FUNCTION_BLOCK FB_HybridDispenser EXTENDS FB_GCodeTool IMPLEMENTS I_Dispenser
VAR_INPUT
END_VAR
VAR_OUTPUT
END_VAR
VAR
	//Specproperties
	aiDispenser		: ARRAY[1..3] OF I_Dispenser;
	nMasterSlotNr	: USINT;

	//****************************************Aktionsvariablen****************************************************
	bBasicDispense			: BOOL;
	nStateA_BasicDispense 	: USINT;
	
	n : INT; //Zählvariablen
	m : INT; //Zählvariablen

END_VAR

IF eCurrentState = E_MachineState.MACHINESTATE_Active THEN
	IF bBasicDispense THEN
		A_HybridDispense();
		IF nStateA_BasicDispense >= 80 THEN
			IF nStateA_BasicDispense >= 99 THEN
				bError := TRUE;
			END_IF
			bBasicDispense := FALSE;
			nStateA_BasicDispense := 0;
			M_RemoveListEntry(nSearchValue:= E_Action.ACTION_BasicDispense);
		END_IF
	END_IF
END_IF

SUPER^();	//FB_MzTool aufrufen

//Prozessdaten aktualisieren
stProcessData.n32Data[7] := BOOL_TO_DINT(bBasicDispense);
aObjProcData[nNotifyId] := stProcessData;

ACTION A_HybridDispense:
IF nStateA_BasicDispense = 0 THEN	//alle Dispenser starten
	FOR n := 1 TO 3 BY 1 DO
		IF aiDispenser[n] <> 0 THEN
			stError.ErrorId := aiDispenser[n].M_DispenserStart();
			stError.ObjectId := aiDispenser[n].P_pObject^.P_nObjectID;
			IF stError.ErrorId > 0 THEN
				//Bereits gestartete Tools wieder stoppen
				FOR m := 1 TO n - 1 BY 1 DO
					aiDispenser[m].M_DispenserStop();
				END_FOR
				nStateA_BasicDispense := 99;
				EXIT;
			END_IF
		END_IF
	END_FOR
	IF nStateA_BasicDispense = 0 THEN
		nStateA_BasicDispense := 1;	
	END_IF
END_IF

IF nStateA_BasicDispense = 1 THEN	//alle Dispenser laufen -> permanent auf Fehler überwachen
	//Das Verlassen dieses States erfolgt durch die Action "HybridDispense" mit Parameter "off" oder durch Stop bzw. Cancel
	FOR n := 1 TO 3 BY 1 DO
		IF aiDispenser[n] <> 0 THEN
			IF aiDispenser[n].P_bError THEN
				stError.ErrorId := aiDispenser[n].P_nErrorId;
				stError.ObjectId := aiDispenser[n].P_pObject^.P_nObjectID;
				nStateA_BasicDispense := 2; //weiter zu stoppen
				EXIT;
			END_IF
		END_IF
	END_FOR	
END_IF

IF nStateA_BasicDispense = 2 THEN //übrige Dispenser nach Fehler stoppen
	nStateA_BasicDispense := 99;
	FOR n := 1 TO 3 BY 1 DO
		IF aiDispenser[n] <> 0 THEN
			IF NOT aiDispenser[n].P_bError THEN
				aiDispenser[n].M_DispenserStop();
			END_IF
		END_IF
	END_FOR	
END_IF

IF nStateA_BasicDispense = 70 THEN //Dispenser stoppen
	nStateA_BasicDispense := 71;
	FOR n := 1 TO 3 BY 1 DO
		IF aiDispenser[n] <> 0 THEN
			aiDispenser[n].M_DispenserStop();
		END_IF
	END_FOR	
ELSIF nStateA_BasicDispense = 71 THEN //warten bis alle Dispenser gestoppt
	nStateA_BasicDispense := 80;
	FOR n := 1 TO 3 BY 1 DO
		IF aiDispenser[n] <> 0 THEN
			IF NOT aiDispenser[n].P_eDispenserState = E_DispenserState.Idle THEN 
				nStateA_BasicDispense := 71;
			END_IF
		END_IF
	END_FOR	
END_IF

//Errorhandling
IF nStateA_BasicDispense = 99 THEN
	stError.Cmd := E_Action.ACTION_BasicDispense;
	stError.POU := E_POU.POU_FB_HybridDispenser;
	stError.POUAction := E_POUACT.POUACT_A_BasicDispense;
	fbErrorList.M_Add(stError);
END_IF
END_ACTION

ACTION A_Reset:
//Ist noch eine Aktion aktiv?
IF nStateA_ResetSpec = 0 THEN 
	(*IF bHeating THEN
		bHeating := FALSE;
		nStateA_Heating := 0;
	END_IF*)
	nStateA_ResetSpec := 80;
END_IF

SUPER^.A_Reset();
END_ACTION

ACTION A_Stop:
IF nStateA_Stop = 0 THEN
	IF bBasicDispense AND nStateA_BasicDispense = 1 THEN
		nStateA_BasicDispense := 70;
	END_IF
	nStateA_Stop := 1;	
END_IF

SUPER^.A_Stop();
END_ACTION

METHOD FB_init : BOOL
VAR_INPUT
	bInitRetains : BOOL; // if TRUE, the retain variables are initialized (warm start / cold start)
	bInCopyCode : BOOL;  // if TRUE, the instance afterwards gets moved into the copy code (online change)
END_VAR
eObjectType := E_ObjectType.OBJECTTYPE_HybridDispenser;
eObjectGroup := E_ObjectGroup.OBJECTGROUP_MzTool OR E_ObjectGroup.OBJECTGROUP_Device;
END_METHOD

METHOD M_AddChild : ERRORID
VAR_INPUT
	pObject : POINTER TO FB_Object;
	nSlotNr	: UINT;
	nIndex : INT;
END_VAR
//Der HybridDispenser kann folgende Objekttypen aufnehmen
//Extruder, PassivePip, CartDispenser
IF pObject > 0 THEN
	IF pObject^.P_eObjectType = E_ObjectType.OBJECTTYPE_Extruder OR
		pObject^.P_eObjectType = E_ObjectType.OBJECTTYPE_CartDispenser OR
		pObject^.P_eObjectType = E_ObjectType.OBJECTTYPE_CartDispStirrer OR
		pObject^.P_eObjectType = E_ObjectType.OBJECTTYPE_PassivPip THEN
		M_AddChild := SUPER^.M_AddChild(pObject,nSlotNr,nIndex);
	ELSE
		M_AddChild := E_ErrorIdObjMgmt.ERRORID_InvalidParentObject;
	END_IF
ELSE
	M_AddChild := E_ErrorIdObjMgmt.ERRORID_InvalidParentObject;
END_IF
END_METHOD

METHOD M_CancelAction
VAR_INPUT
	eAction : E_Action;
END_VAR
CASE eAction OF
	E_Action.ACTION_BasicDispense:
		IF bBasicDispense AND nStateA_BasicDispense = 1 THEN
			nStateA_BasicDispense := 70;
		END_IF
ELSE
	SUPER^.M_CancelAction(eAction);
END_CASE
END_METHOD

METHOD M_CheckAction : ERRORID
VAR_INPUT
	refActionData 	: REFERENCE TO ST_ActionData;
	pCorrelObject	: POINTER TO FB_Object;
END_VAR
CASE refActionData.eAction OF
	E_Action.ACTION_Dispense,
	E_Action.ACTION_CleanTip,
	E_Action.ACTION_MeasureTool,
	E_Action.ACTION_TeachTarget:
		RETURN;
ELSE
	M_CheckAction := SUPER^.M_CheckAction(refActionData, pCorrelObject);
END_CASE
END_METHOD

METHOD M_CheckGCodeStart : ERRORID
VAR_INPUT
END_VAR

VAR
	i : USINT;
	pGCodeTool : POINTER TO FB_GCodeTool;
END_VAR
FOR i := 1 TO 3 BY 1 DO
	IF aiDispenser[i] <> 0 AND_THEN aiDispenser[i].P_pObject^.P_eObjectType = E_ObjectType.OBJECTTYPE_Extruder THEN
		pGCodeTool := aiDispenser[i].P_pObject;
		M_CheckGCodeStart := pGCodeTool^.M_CheckGCodeStart();
		IF M_CheckGCodeStart > 0 THEN
			RETURN;
		END_IF
	END_IF
END_FOR
END_METHOD

METHOD M_CheckProcDataType : BOOL
VAR_INPUT
	eProcDataType : E_ProcDataType;
END_VAR
END_METHOD

METHOD M_CheckProps : ERRORID
VAR_INPUT
END_VAR

VAR
	i 				: UINT;
	pSlot 			: POINTER TO FB_Slot;
	pExtruder 		: POINTER TO FB_Extruder;
	pCartDispenser 	: POINTER TO FB_CartDispenser;
	pPassivePip 	: POINTER TO FB_PassivPip;
END_VAR
M_CheckProps := SUPER^.M_CheckProps();
//Kann bis zu 3 CartDispenser enthalten
aiDispenser[1] := 0;
aiDispenser[2] := 0;
aiDispenser[3] := 0;
FOR i:= 1 TO nNumberOfSlots BY 1 DO
	pSlot := fbSlotList.M_GetAtNr(i);
	IF pSlot > 0 AND_THEN pSlot^.P_pChild > 0  THEN
		//Achtung, nur Tools die das Interface "I_HybridDispenser" implementieren sind erlaubt!
		IF pSlot^.P_pChild^.P_eObjectType = E_ObjectType.OBJECTTYPE_Extruder THEN
			pExtruder := pSlot^.P_pChild;
			aiDispenser[pSlot^.P_nNr] := pExtruder^;
		ELSIF pSlot^.P_pChild^.P_eObjectType = E_ObjectType.OBJECTTYPE_CartDispenser OR 
				pSlot^.P_pChild^.P_eObjectType = E_ObjectType.OBJECTTYPE_CartDispStirrer THEN
			pCartDispenser := pSlot^.P_pChild;
			aiDispenser[pSlot^.P_nNr] := pCartDispenser^;
		ELSIF pSlot^.P_pChild^.P_eObjectType = E_ObjectType.OBJECTTYPE_PassivPip THEN
			pPassivePip := pSlot^.P_pChild;
			aiDispenser[pSlot^.P_nNr] := pPassivePip^;
		END_IF
	END_IF
END_FOR
//MasterSlotNr auswerten
//1. kann nur 1,2 oder 3 sein
//2. entsprechender Slot muss belegt sein
IF nMasterSlotNr >= 1 AND nMasterSlotNr <= 3 THEN
	IF aiDispenser[nMasterSlotNr] = 0 THEN
		M_CheckProps := E_ErrorIdObjMgmt.ERRORID_NoToolOnMasterSlot;	
	END_IF
ELSE
	M_CheckProps := E_ErrorIdObjMgmt.ERRORID_InvalidSlotNumber;
END_IF
END_METHOD

METHOD M_ClearAllProps
VAR_INPUT
	bIgnoreParent : BOOL; //Es wird das gesamte OD gelöscht. -> Zeiger auf Parent nicht mehr gültig!
END_VAR
aiDispenser[1] := 0;
aiDispenser[2] := 0;
aiDispenser[3] := 0;
SUPER^.M_ClearAllProps(bIgnoreParent);
END_METHOD

METHOD M_DispenserPrepare : ERRORID
VAR_INPUT
END_VAR
//do nothing
END_METHOD

METHOD M_DispenserStart : ERRORID
VAR_INPUT
END_VAR
IF NOT (eCurrentState = E_MachineState.MACHINESTATE_Idle OR
	eCurrentState = E_MachineState.MACHINESTATE_Active OR
	eCurrentState = E_MachineState.MACHINESTATE_Ready) THEN
	M_DispenserStart := E_ErrorIdCmd.ERRORID_InvalidState;
	RETURN;
END_IF
			
IF NOT bBasicDispense THEN
	bBasicDispense := TRUE;
	fbList.A_AddHeadValue(hList := hList, putValue := E_Action.ACTION_BasicDispense);
ELSE //Bereits Ein -> Error werfen
	M_DispenserStart := E_ErrorIdCmd.ERRORID_BasicActionActive;
	RETURN;
END_IF

bBusy := TRUE;
eCurrentState := E_MachineState.MACHINESTATE_Active;
END_METHOD

METHOD M_DispenserStop : ERRORID
VAR_INPUT
END_VAR
IF bBasicDispense AND nStateA_BasicDispense = 1 THEN
	nStateA_BasicDispense := 70;
END_IF
END_METHOD

METHOD M_ExeAction : ERRORID
VAR_INPUT
	refActionData : REFERENCE TO ST_ActionData;	
END_VAR
IF NOT (eCurrentState = E_MachineState.MACHINESTATE_Idle OR
	eCurrentState = E_MachineState.MACHINESTATE_Active OR
	eCurrentState = E_MachineState.MACHINESTATE_Ready) THEN
	M_ExeAction := E_ErrorIdCmd.ERRORID_InvalidState;
	RETURN;
END_IF

CASE refActionData.eAction OF
	E_Action.ACTION_BasicDispense:
		IF refActionData.aParams[1] = 0 THEN //Aus
			M_ExeAction := M_DispenserStop();
		ELSE //Ein
			M_ExeAction := M_DispenserStart();
		END_IF
	ELSE
		M_ExeAction := SUPER^.M_ExeAction(refActionData);
		RETURN;
END_CASE
END_METHOD

METHOD M_GetAllProps : ERRORID
VAR_INPUT
	refCmdData : REFERENCE TO  ST_CmdData;
END_VAR
SUPER^.M_GetAllProps(refCmdData);
nCurrentPropIndex := nCurrentPropIndex + 1;
refCmdData.n32Data[nCurrentPropIndex] := nMasterSlotNr;
END_METHOD

METHOD M_GetNozzle : POINTER TO FB_Nozzle
VAR_INPUT
END_VAR
IF P_pMasterTool > 0 THEN
	M_GetNozzle := P_pMasterTool^.M_GetNozzle();
END_IF
END_METHOD

METHOD M_GetProcData : DINT
VAR_INPUT
	eProcDataType : E_ProcDataType;
END_VAR
END_METHOD

METHOD M_GetZAxisRef : POINTER TO FB_ZAxisRef
VAR_INPUT
	pTool : POINTER TO FB_MzTool;
	pToolSlot : POINTER TO FB_Slot;
END_VAR

VAR
	nSlotDiff : INT;
	nAxisNr : INT;
END_VAR
//Diese Methode überschreibt sie Methode von FB_MzTool und wird derzeit nur vom SyringeExtruder (Child) aufgerufen
IF pTool^.P_eObjectType = E_ObjectType.OBJECTTYPE_Extruder THEN
	nSlotDiff :=  UINT_TO_INT(pToolSlot^.P_nNr) - UINT_TO_INT(nMasterSlotNr);
	nAxisNr := pZAxisRef^.nChannel + nSlotDiff * 2; //Es muss immer eine freie Achse dazwischen sein.
	M_GetZAxisRef := ADR(pFbMultiZ^.aFbZAxisRef[nAxisNr]);
	IF M_GetZAxisRef^.eDetectedToolType <> E_MzToolType.TOOL_TYPE_SyringeExtruder THEN
		M_GetZAxisRef := 0;
	END_IF
ELSE
	M_GetZAxisRef := SUPER^.M_GetZAxisRef(pTool, pParentSlot);
END_IF
END_METHOD

METHOD M_Prepare : ST_MethResult
VAR_INPUT
	bExecute : BOOL;
END_VAR

VAR
 	i : USINT;	
END_VAR

VAR_INST
	nState : USINT;	
END_VAR
IF bExecute THEN
	IF nState = 0 THEN
		nState := 80;
		FOR i := 1 TO 3 BY 1 DO
			IF aiDispenser[i] <> 0 THEN
				M_Prepare.nErrorId := aiDispenser[i].M_DispenserPrepare();
				IF M_Prepare.nErrorId > 0 THEN
					M_Prepare.bError := TRUE;
					M_Prepare.bBusy := FALSE;
					RETURN;
				END_IF
				IF aiDispenser[i].P_eDispenserState = E_DispenserState.Preparing THEN
					nState := 1;
					M_Prepare.bBusy := TRUE;				
					RETURN;
				END_IF
			END_IF
		END_FOR
	ELSIF nState = 1 THEN
		FOR i := 1 TO 3 BY 1 DO
			IF aiDispenser[i] <> 0 THEN
				IF aiDispenser[i].P_bError THEN
					M_Prepare.bError := TRUE;
					M_Prepare.bBusy := FALSE;
					RETURN;
				END_IF
				IF aiDispenser[i].P_eDispenserState = E_DispenserState.Preparing THEN
					nState := 1;
					M_Prepare.bBusy := TRUE;
					RETURN;
				END_IF				
			END_IF
		END_FOR
	END_IF
ELSE
	nState := 0;	
END_IF
END_METHOD

METHOD M_SetAllProps : ERRORID
VAR_INPUT
	refCmdData : REFERENCE TO  ST_CmdData;
END_VAR
M_SetAllProps := SUPER^.M_SetAllProps(refCmdData);

IF M_SetAllProps > 0 THEN
	RETURN;
END_IF

nCurrentPropIndex := nCurrentPropIndex + 1;
nSpecPropIndex := nCurrentPropIndex;
nMasterSlotNr := DINT_TO_USINT(refCmdData.n32Data[nCurrentPropIndex]);
nNoOfProps := nCurrentPropIndex + 1;
END_METHOD

METHOD M_SetPrintParams : ST_MethResult
VAR_INPUT
	eType 		: E_PrintParamType;
	nNumerator	: USINT;
	nValue		: DINT;
END_VAR

VAR
	pGCodeTool		: POINTER TO FB_GCodeTool;
END_VAR
CASE eType OF
	E_PrintParamType.Pressure:
		CASE nNumerator OF
			1:	IF aiDispenser[1] <> 0 AND_THEN 
					(aiDispenser[1].P_pObject^.P_eObjectType = E_ObjectType.OBJECTTYPE_CartDispenser OR	aiDispenser[1].P_pObject^.P_eObjectType = E_ObjectType.OBJECTTYPE_CartDispStirrer) THEN
					pGCodeTool := aiDispenser[1].P_pObject;
					M_SetPrintParams := pGCodeTool^.M_SetPrintParams(E_PrintParamType.Pressure, 1, nValue);
				ELSE
					M_SetPrintParams.bError := TRUE;
					M_SetPrintParams.nErrorId := E_ErrorIdCmd.ERRORID_InvalidPrintParamType;
				END_IF
				
			2:	IF aiDispenser[2] <> 0 AND_THEN
					(aiDispenser[2].P_pObject^.P_eObjectType = E_ObjectType.OBJECTTYPE_CartDispenser OR aiDispenser[2].P_pObject^.P_eObjectType = E_ObjectType.OBJECTTYPE_CartDispStirrer) THEN
					pGCodeTool := aiDispenser[2].P_pObject;
					M_SetPrintParams := pGCodeTool^.M_SetPrintParams(E_PrintParamType.Pressure, 1, nValue);
				ELSE
					M_SetPrintParams.bError := TRUE;
					M_SetPrintParams.nErrorId := E_ErrorIdCmd.ERRORID_InvalidPrintParamType;
				END_IF
			
			3: IF aiDispenser[3] <> 0 AND_THEN
					(aiDispenser[3].P_pObject^.P_eObjectType = E_ObjectType.OBJECTTYPE_CartDispenser OR aiDispenser[3].P_pObject^.P_eObjectType = E_ObjectType.OBJECTTYPE_CartDispStirrer) THEN
					pGCodeTool := aiDispenser[3].P_pObject;
					M_SetPrintParams := pGCodeTool^.M_SetPrintParams(E_PrintParamType.Pressure, 1, nValue);
				ELSE
					M_SetPrintParams.bError := TRUE;
					M_SetPrintParams.nErrorId := E_ErrorIdCmd.ERRORID_InvalidPrintParamType;
				END_IF
		ELSE
			M_SetPrintParams.bError := TRUE;
			M_SetPrintParams.nErrorId := E_ErrorIdCmd.ERRORID_InvalidPrintParamNumerator;
		END_CASE
		
	E_PrintParamType.Feed:
		CASE nNumerator OF
			1:	IF aiDispenser[1] <> 0 AND_THEN aiDispenser[1].P_pObject^.P_eObjectType = E_ObjectType.OBJECTTYPE_Extruder THEN
					pGCodeTool := aiDispenser[1].P_pObject;
					M_SetPrintParams := pGCodeTool^.M_SetPrintParams(E_PrintParamType.Feed, 1, nValue);
				ELSE
					M_SetPrintParams.bError := TRUE;
					M_SetPrintParams.nErrorId := E_ErrorIdCmd.ERRORID_InvalidPrintParamType;
				END_IF
			
			2:	IF aiDispenser[2] <> 0 AND_THEN aiDispenser[2].P_pObject^.P_eObjectType = E_ObjectType.OBJECTTYPE_Extruder THEN
					pGCodeTool := aiDispenser[2].P_pObject;
					M_SetPrintParams := pGCodeTool^.M_SetPrintParams(E_PrintParamType.Feed, 1, nValue);
				ELSE
					M_SetPrintParams.bError := TRUE;
					M_SetPrintParams.nErrorId := E_ErrorIdCmd.ERRORID_InvalidPrintParamType;
				END_IF
			
			3:	IF aiDispenser[3] <> 0 AND_THEN aiDispenser[3].P_pObject^.P_eObjectType = E_ObjectType.OBJECTTYPE_Extruder THEN
					pGCodeTool := aiDispenser[3].P_pObject;
					M_SetPrintParams := pGCodeTool^.M_SetPrintParams(E_PrintParamType.Feed, 1, nValue);			
				ELSE
					M_SetPrintParams.bError := TRUE;
					M_SetPrintParams.nErrorId := E_ErrorIdCmd.ERRORID_InvalidPrintParamType;
				END_IF
			
		ELSE
			M_SetPrintParams.bError := TRUE;
			M_SetPrintParams.nErrorId := E_ErrorIdCmd.ERRORID_InvalidPrintParamNumerator;
		END_CASE
		
	E_PrintParamType.Flow:
		CASE nNumerator OF
			1:	IF aiDispenser[1] <> 0 AND_THEN aiDispenser[1].P_pObject^.P_eObjectType = E_ObjectType.OBJECTTYPE_PassivPip THEN
					pGCodeTool := aiDispenser[1].P_pObject;
					M_SetPrintParams := pGCodeTool^.M_SetPrintParams(E_PrintParamType.Flow, 1, nValue);			
				ELSE
					M_SetPrintParams.bError := TRUE;
					M_SetPrintParams.nErrorId := E_ErrorIdCmd.ERRORID_InvalidPrintParamType;
				END_IF
			
			2:	IF aiDispenser[2] <> 0 AND_THEN aiDispenser[2].P_pObject^.P_eObjectType = E_ObjectType.OBJECTTYPE_PassivPip THEN
					pGCodeTool := aiDispenser[2].P_pObject;
					M_SetPrintParams := pGCodeTool^.M_SetPrintParams(E_PrintParamType.Flow, 1, nValue);			
				ELSE
					M_SetPrintParams.bError := TRUE;
					M_SetPrintParams.nErrorId := E_ErrorIdCmd.ERRORID_InvalidPrintParamType;
				END_IF
			
			3:	IF aiDispenser[3] <> 0 AND_THEN aiDispenser[3].P_pObject^.P_eObjectType = E_ObjectType.OBJECTTYPE_PassivPip THEN
					pGCodeTool := aiDispenser[3].P_pObject;
					M_SetPrintParams := pGCodeTool^.M_SetPrintParams(E_PrintParamType.Flow, 1, nValue);
				ELSE
					M_SetPrintParams.bError := TRUE;
					M_SetPrintParams.nErrorId := E_ErrorIdCmd.ERRORID_InvalidPrintParamType;
				END_IF
		ELSE
			M_SetPrintParams.bError := TRUE;
			M_SetPrintParams.nErrorId := E_ErrorIdCmd.ERRORID_InvalidPrintParamNumerator;
		END_CASE
	
ELSE
	M_SetPrintParams.bError := TRUE;
	M_SetPrintParams.nErrorId := E_ErrorIdCmd.ERRORID_InvalidPrintParamType;	
END_CASE
END_METHOD

METHOD M_ToolIsOnMasterSlot : BOOL
VAR_INPUT
	pTool : POINTER TO FB_MzTool;
END_VAR
IF aiDispenser[nMasterSlotNr] <> 0 THEN
	M_ToolIsOnMasterSlot := aiDispenser[nMasterSlotNr].P_pObject = pTool;
END_IF
END_METHOD

PROPERTY P_bSensorMounted : BOOL
GET
VAR
	i : USINT;
	pTool : POINTER TO FB_MzTool;
END_VAR
FOR i := 1 TO 3 BY 1 DO
	IF aiDispenser[i] <> 0 THEN
		pTool := aiDispenser[i].P_pObject;
		IF pTool^.P_bSensorMounted THEN
			P_bSensorMounted := TRUE;
			RETURN;
		END_IF
	END_IF
END_FOR
END_GET
END_PROPERTY

PROPERTY P_eDispenserState : E_DispenserState
GET
IF bBasicDispense THEN
	//falls ein Dispenser in Preparing ist, dann bleibt es auch so
	P_eDispenserState := E_DispenserState.Dispensing;
END_IF
END_GET
END_PROPERTY

PROPERTY P_pMasterTool : POINTER TO FB_MzTool
GET
P_pMasterTool := aiDispenser[nMasterSlotNr].P_pObject;
END_GET
END_PROPERTY

PROPERTY P_stAbsPosPhys : ST_3DPoint
GET
VAR
	pMzTool : POINTER TO FB_MzTool;
END_VAR
IF aiDispenser[nMasterSlotNr] <> 0 THEN
	pMzTool := aiDispenser[nMasterSlotNr].P_pObject;
	P_stAbsPosPhys := pMzTool^.P_stAbsPosPhys;
ELSE
	P_stAbsPosPhys := SUPER^.P_stAbsPosPhys;
END_IF
END_GET
END_PROPERTY

END_FUNCTION_BLOCK

(* stored: Version 1.1.0.1, ProductVersion 3.1.4024.9
   POU FB_HybridDispenser: Id {66f767df-9f17-4ced-a0df-52e824ae2671}, SpecialFunc None
   Action A_HybridDispense: Id {8d936772-d544-4aa1-b19b-e969ff87b9cd}
   Action A_Reset: Id {a482625e-95ff-4fc4-a8cf-cf30f2fadff5}
   Action A_Stop: Id {89cdf597-595e-4299-9c5d-649fedd30289}
   Method FB_init: Id {2333ea12-39e9-4cf7-bea4-0fef2cd95c61}
   Method M_AddChild: Id {7f082068-4121-4e0b-b214-b6ed87056bd0}
   Method M_CancelAction: Id {0eb8483b-a2c5-4a27-8b71-cdc358ad185a}
   Method M_CheckAction: Id {3cce8f03-648c-4a92-a172-ac413395076f}
   Method M_CheckGCodeStart: Id {530f3c3b-309f-4d22-b9c7-d04106859303}
   Method M_CheckProcDataType: Id {ffc69ed7-3e8a-4196-8a81-99fce50d3127}
   Method M_CheckProps: Id {8bfd8b2d-e3c6-4785-a17a-f0537452959e}
   Method M_ClearAllProps: Id {8920eafd-edd7-4aba-9df0-5e19972f99e9}
   Method M_DispenserPrepare: Id {2fc4be12-cb16-4947-9f14-9c42df44b7e5}
   Method M_DispenserStart: Id {90b2ab18-a6a9-473a-86a5-e8c5651168e4}
   Method M_DispenserStop: Id {99c96599-5de0-44af-985a-e499f40f70e6}
   Method M_ExeAction: Id {e570641e-3944-4e20-a230-a7e777f8d928}
   Method M_GetAllProps: Id {0ade4717-60a7-43c1-a3b2-f1d00a3babc7}
   Method M_GetNozzle: Id {54003e9d-1a7e-4518-9f82-a0e4bed7ffa2}
   Method M_GetProcData: Id {b91c04bd-1aaf-4af8-ac63-dcb82cd99d8e}
   Method M_GetZAxisRef: Id {1218632a-890c-4c63-be50-c700c3f80add}
   Method M_Prepare: Id {66ee8406-4dd6-4e43-a22f-1912ca01857b}
   Method M_SetAllProps: Id {d76f5aa1-fc0f-4796-96ae-7d0ae9669b6e}
   Method M_SetPrintParams: Id {97f76bc7-a6d8-4827-b068-a6c6aae97478}
   Method M_ToolIsOnMasterSlot: Id {8d748c99-386e-4952-9a33-6e5d28b55d4f}
   Property P_bSensorMounted: Id {c961256e-9310-4dd8-80f5-ab8fb1f9164e}
   Get Get: Id {83023f0a-84ac-4614-93f5-de90902b0709}
   Property P_eDispenserState: Id {deb289a2-725e-4a6e-be13-6d6c9b05232f}
   Get Get: Id {e212129a-ab1c-4bef-873c-92ba9aa69152}
   Property P_pMasterTool: Id {630fdeaa-fa3b-4de2-a160-0f7c814075f0}
   Get Get: Id {8fe4ec90-7ed9-444e-ac0c-3e8bfbf4077b}
   Property P_stAbsPosPhys: Id {433a5fc6-1111-403e-ade2-9ac65768d9e2}
   Get Get: Id {a5246394-6913-468b-9907-2dff676decc7} *)
